FUNCTION_BLOCK FB_SIM_ACTUATOR
VAR_INPUT
	ptrDev:		POINTER TO FB_ACTUATOR;
END_VAR
VAR_OUTPUT
END_VAR
VAR
	{attribute 'OPC.UA.DA':='0'}
	ptrCfg:		POINTER TO T_ACTUATOR_CFG;
	{attribute 'OPC.UA.DA':='0'}
	ptrStat:	POINTER TO T_ACTUATOR_STAT;

	{attribute 'OPC.UA.DA':='1'}
	cfg:			T_SIM_ACTUATOR_CFG;		(* ActiveLow configuration for each signal *)
	{attribute 'OPC.UA.DA':='1'}
	stat:			T_SIM_ACTUATOR_STAT;	(* Simulator status parameters *)
	
	{attribute 'OPC.UA.DA':='0'}
	bSwitch:		BOOL := FALSE;
	{attribute 'OPC.UA.DA':='0'}
	bSwitchLast:	BOOL := FALSE;
	
	{attribute 'OPC.UA.DA':='0'}
	bOn:			BOOL := TRUE;
	{attribute 'OPC.UA.DA':='0'}
	nCouplerState:	UINT := 8;       // normal coupler state
	
    (* Inputs *)
	{attribute 'OPC.UA.DA':='0'}
	i_bSwitch 		AT %I*: 	BOOL;

	(* Outputs *)	
	{attribute 'OPC.UA.DA':='0'}
	q_bOn 		AT %Q*: 		BOOL;
	{attribute 'OPC.UA.DA':='0'}
	q_nCouplerState AT %Q*:		UINT := 8;
	
	{attribute 'OPC.UA.DA':='0'}
	timer:			TON;
	
	{attribute 'OPC.UA.DA':='0'}
	trigger:		R_TRIG;	// To capture device INIT
	
END_VAR

IF NOT stat.bInitialised THEN
	ptrCfg	:= ADR(ptrDev^.cfg);
	ptrStat	:= ADR(ptrDev^.stat);

	// Check for NULL pointers in input parameters
	IF ptrCfg = 0  OR  ptrStat = 0 THEN
		stat.nErrorCode	:= E_ACTUATOR_ERROR.ZERO_POINTER;
		stat.sErrorText	:= 'ERROR: Input parameter is a NULL pointer';
		stat.sStatus	:= 'ERROR';
		RETURN;
	END_IF

	RPC_ResetConfig();	// Copy configuration from device
	
	timer(IN:=FALSE);
	timer(IN:=TRUE,PT:=UDINT_TO_TIME(100));	// Update almost immediately

	stat.nErrorCode	:= E_ACTUATOR_ERROR.OK;
	stat.sErrorText	:= 'OK';
	stat.sStatus	:= 'OK';
	
	stat.bInitialised	:= TRUE;
	RETURN;
END_IF

// There are two triggers: 
// 	Detect device INIT
// 	Activation of switch

// Check for INIT trigger
//trigger(CLK:=(ptrStat^.sActionDesc = 'ActionInitExecute'));
trigger(CLK:=(	ptrStat^.nSubstate=E_ACTUATOR_SUBSTATE.NOTOP_SWITCHING_ON OR 
				ptrStat^.nSubstate=E_ACTUATOR_SUBSTATE.NOTOP_SWITCHING_OFF));

// Get the state of control command
bSwitch := GetLogicalState(i_bSwitch, cfg.bActiveLowSwitch);

IF trigger.Q THEN
	RPC_ResetConfig();	// Copy configuration from device
ELSIF bSwitch <> bSwitchLast THEN
	// Switch value has changed. 
	bSwitchLast	:= bSwitch;
	// Delayed response
	timer(IN:=FALSE);
	timer(IN:=TRUE,PT:=UDINT_TO_TIME(cfg.nDelay));
END_IF


// Execute the timer
timer();

// Set new outputs once the timer has expired
IF timer.Q THEN
	timer(IN:=FALSE);	// Reset timer
	// Set output, i.e. feedback
	bOn	:= GetLogicalState(bSwitch,	cfg.bActiveLowOn);
END_IF


(* Assign outputs *)
q_bOn 			:= bOn;
q_nCouplerState := nCouplerState;

METHOD GetLogicalState : BOOL
(*
	This method returns the state of the variable based on its 
	activeLow configuration.
	Syntax:
		bState	:= GetLogicalState (<var value>,  <activeLow cfg>);
		
	Example 1:
		var = TRUE;
		activeLow = FALSE;
		bState	:= GetLogicalState (TRUE,  FALSE); = TRUE

	Example 2:
		var = TRUE;
		activeLow = TRUE;
		bState	:= GetLogicalState (TRUE,  TRUE); = FALSE
*)
VAR_INPUT
	state:		BOOL;
	activeLow:	BOOL;
END_VAR
IF activeLow THEN
	GetLogicalState := NOT state;
ELSE
	GetLogicalState := state;
END_IF
END_METHOD

{attribute 'TcRpcEnable':='1'}
METHOD RPC_ResetConfig : BOOL
VAR_INPUT
END_VAR
cfg.bActiveLowOn		:= ptrCfg^.bActiveLowOn;
cfg.bActiveLowSwitch	:= ptrCfg^.bActiveLowSwitch;
// Response delay = 1/2 of real switch timeout - the stable signal period
cfg.nDelay				:= ptrCfg^.nTimeout / 2 - ptrCfg^.nSigStablePeriod;	
IF cfg.nDelay < 0 THEN
	cfg.nDelay	:= 0;
END_IF
nCouplerState			:= 8;

// Get the Switch value
bSwitch := GetLogicalState(i_bSwitch, cfg.bActiveLowSwitch);

bOn	:= GetLogicalState(bSwitch,	cfg.bActiveLowOn);	// Set Switch state

RPC_ResetConfig	:= TRUE;
END_METHOD

{attribute 'TcRpcEnable':='1'}
METHOD RPC_SetActiveLow_On : BOOL
VAR_INPUT
	bValue:	BOOL;
END_VAR
cfg.bActiveLowOn	:= bValue;

RPC_SetActiveLow_On	:= TRUE;
END_METHOD

{attribute 'TcRpcEnable':='1'}
METHOD RPC_SetActiveLow_Switch : BOOL
VAR_INPUT
	bValue:	BOOL;
END_VAR
cfg.bActiveLowSwitch	:= bValue;

RPC_SetActiveLow_Switch	:= TRUE;
END_METHOD

{attribute 'TcRpcEnable':='1'}
METHOD RPC_SetCouplerState : BOOL
VAR_INPUT
	bValue:	UINT;
END_VAR
nCouplerState	:= bValue;

RPC_SetCouplerState	:= TRUE;
END_METHOD

{attribute 'TcRpcEnable':='1'}
METHOD RPC_SetDelay : BOOL
VAR_INPUT
	nDelay:	UDINT;	// Response delay [msec]
END_VAR
cfg.nDelay	:= nDelay;

RPC_SetDelay	:= TRUE;
END_METHOD

END_FUNCTION_BLOCK

(* stored: Version 1.1.0.1, ProductVersion 3.1.4024.3
   POU FB_SIM_ACTUATOR: Id {cdc20ae3-b7e8-4041-8913-f51782748d05}, SpecialFunc None
   Method GetLogicalState: Id {3a675f1a-7819-414a-ae93-030e56ccbed7}
   Method RPC_ResetConfig: Id {cefd105e-0777-45a9-b272-dea41c909353}
   Method RPC_SetActiveLow_On: Id {23934f2f-e237-4c2f-ac22-9cf7b73719c4}
   Method RPC_SetActiveLow_Switch: Id {a4ecdb8e-bcef-4dcf-b895-66561c234cd6}
   Method RPC_SetCouplerState: Id {45255316-3d56-412d-a07e-b4d5796053d0}
   Method RPC_SetDelay: Id {1004106a-d14c-4cdf-9cbe-1c39692b430f} *)
